TYPE TFMachinePalletizer_LatoApprendimento :
STRUCT
	Lato0 	: TFMachinePalletizer_ApprendimentoQuota;	
	Lato90 	: TFMachinePalletizer_ApprendimentoQuota;
	Lato180 : TFMachinePalletizer_ApprendimentoQuota;
END_STRUCT
END_TYPE

(* stored: Version 1.1.0.1, ProductVersion 3.1.4024.11
   DUT TFMachinePalletizer_LatoApprendimento: Id {3b0569ea-90f3-4416-9f40-bcd7097f02f5} *)
